// TIA Portal V16 export
// export: Created 2021-11-12T13:31:40.7607488Z, ExportSetting WithDefaults, DisplayName Totally Integrated Automation Portal, DisplayVersion V16 Update 3, DisplayName TIA Portal Version Control Interface, DisplayVersion V16 Update 2, DisplayName TIA Portal Openness, DisplayVersion V16 Update 3, DisplayName SINAMICS Startdrive Advanced, DisplayVersion V16 Update 5, DisplayName SINAMICS Startdrive G130, G150, S120, S150, SINAMICS MV, S210, DisplayVersion V16 Update 5, DisplayName SINAMICS Startdrive G110M, G120, G120C, G120D, G120P, G115D, DisplayVersion V16 Update 5, DisplayName STEP 7 Professional, DisplayVersion V16 Update 3, DisplayName STEP 7 Safety, DisplayVersion V16, DisplayName WinCC UA Professional, DisplayVersion V16 Update 3
FUNCTION "MTS_Move" : Void   // FC10, LAD
TITLE = Move material data
{ S7_Optimized_Access := 'TRUE' }
VERSION : 0.1
// Move material data from source position to destination position
// stored: AutoNumber true, IsIECCheckEnabled false, SetENOAutomatically false, UDAEnableTagReadback false
   VAR_OUTPUT
      OS_Destination : "UDT_MatCard";   // Destination data
   END_VAR
   VAR_IN_OUT
      XS_Source : "UDT_MatCard";   // Source data
   END_VAR
BEGIN

REGION Network 1: Copy material data and clear source
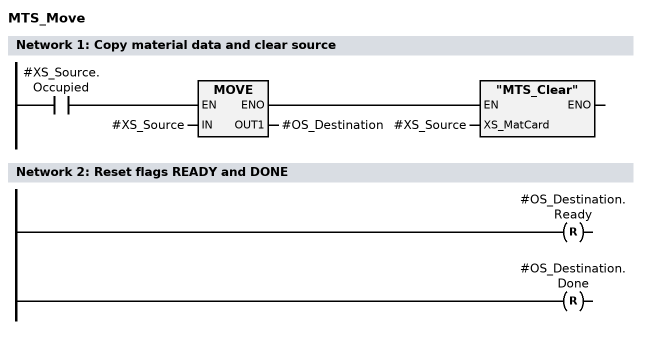
   RUNG wire#powerrail
      Contact( #XS_Source.Occupied )
      Move(in := #XS_Source, out1 => #OS_Destination)
      "MTS_Clear"(XS_MatCard := #XS_Source)
   END_RUNG
   // the same network as SCL:
   IF #XS_Source.Occupied THEN
       #OS_Destination := #XS_Source;
       "MTS_Clear"(XS_MatCard := #XS_Source);
   END_IF;
END_REGION

REGION Network 2: Reset flags READY and DONE
   RUNG wire#powerrail
      R_Coil( #OS_Destination.Ready )
   END_RUNG
   RUNG wire#powerrail
      R_Coil( #OS_Destination.Done )
   END_RUNG
   // the same network as SCL:
   #OS_Destination.Ready := FALSE;
   #OS_Destination.Done := FALSE;
END_REGION
END_FUNCTION
